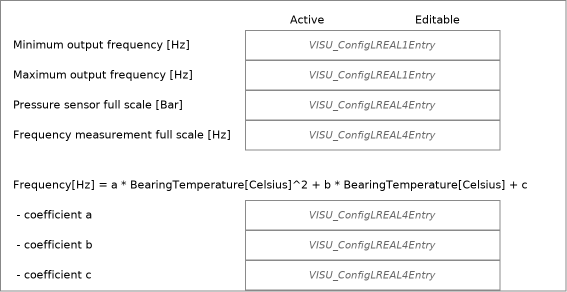
VISUALIZATION VISU_HydraulicsConfig_Side_General  // 567x292
VAR_IN_OUT
    editable : HydraulicsSideConfig;
	active : HydraulicsSideConfig;
END_VAR
    Label (245,10 125x20), "Active"
    Label (375,10 125x20), "Editable"
    Label (10,30 250x30), "Minimum output frequency [Hz]"
    Label (10,60 235x30), "Maximum output frequency [Hz]"
    Frame (245,30 255x30), tooltip "Time (in seconds) to wait after the axis has been moved"
        shows VISU_ConfigLREAL1Entry(active := active.minFrequency, editable := editable.minFrequency)
    Frame (245,60 255x30), tooltip "Time (in seconds) to wait after the axis has been moved"
        shows VISU_ConfigLREAL1Entry(active := active.maxFrequency, editable := editable.maxFrequency)
    Label (10,90 265x30), "Pressure sensor full scale [Bar]"
    Frame (245,90 255x30), tooltip "Time (in seconds) to wait after the axis has been moved"
        shows VISU_ConfigLREAL4Entry(active := active.pressureSensorFullScale, editable := editable.pressureSensorFullScale)
    Label (10,120 265x30), "Frequency measurement full scale [Hz]"
    Frame (245,120 255x30), tooltip "Time (in seconds) to wait after the axis has been moved"
        shows VISU_ConfigLREAL4Entry(active := active.frequencyMeasurementFullScale, editable := editable.frequencyMeasurementFullScale)
    Label (10,200 265x30), "- coefficient a"
    Frame (245,200 255x30), tooltip "Time (in seconds) to wait after the axis has been moved"
        shows VISU_ConfigLREAL4Entry(active := active.conversionCoefficientA, editable := editable.conversionCoefficientA)
    Label (10,230 265x30), "- coefficient b"
    Frame (245,230 255x30), tooltip "Time (in seconds) to wait after the axis has been moved"
        shows VISU_ConfigLREAL4Entry(active := active.conversionCoefficientB, editable := editable.conversionCoefficientB)
    Label (10,260 265x30), "- coefficient c"
    Frame (245,260 255x30), tooltip "Time (in seconds) to wait after the axis has been moved"
        shows VISU_ConfigLREAL4Entry(active := active.conversionCoefficientC, editable := editable.conversionCoefficientC)
    Label (10,170 555x30), "Frequency[Hz] = a * BearingTemperature[Celsius]^2 + b * BearingTemperature[Celsius] + c"
END_VISUALIZATION

(* stored: Version 1.1.0.1, ProductVersion 3.1.4019.2
   Visu VISU_HydraulicsConfig_Side_General: Id {e8f56c23-5357-45c2-8c1a-1b99aefc4a4e} *)
